FUNCTION Convert_LREAL_TO_UINT : Hresult
VAR_INPUT
	in : LREAL;
	out : REFERENCE TO UINT;
END_VAR
VAR
	converted : UINT;
END_VAR
VAR CONSTANT
	INCOMPATIBLE : HRESULT := 16#9811070E;
END_VAR

converted := LREAL_TO_UINT(in);

IF (UINT_TO_LREAL(converted) <> in) THEN
	Convert_LREAL_TO_UINT := INCOMPATIBLE;
	RETURN;
END_IF

out := converted;

END_FUNCTION

(* stored: Version 1.1.0.1, ProductVersion 3.1.4024.12
   POU Convert_LREAL_TO_UINT: Id {ac74376d-8743-4f9a-aaec-25ef03f606bb}, SpecialFunc None *)
